// TIA Portal V20 export
FUNCTION "Level_Sim" : Void   // FC1, FBD
{ S7_Optimized_Access := 'TRUE' }
// stored: SetENOAutomatically false
BEGIN

REGION Network 1: LevelSimulation
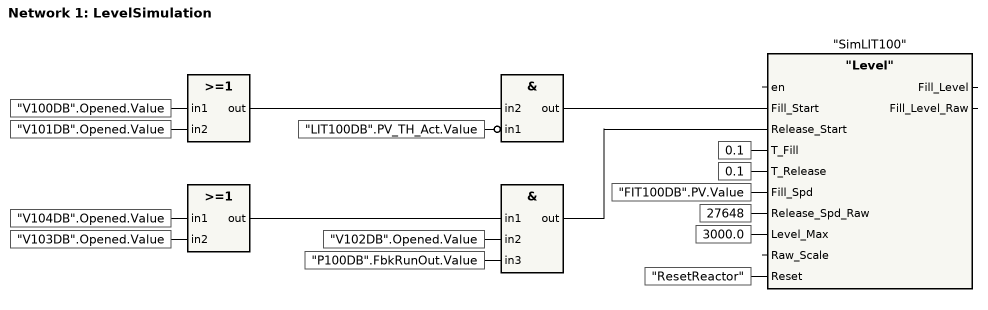
   "SimLIT100"(Fill_Start := ("V100DB".Opened.Value OR "V101DB".Opened.Value) AND NOT "LIT100DB".PV_TH_Act.Value,   // "Level"
               Release_Start := ("V104DB".Opened.Value OR "V103DB".Opened.Value) AND "V102DB".Opened.Value AND "P100DB".FbkRunOut.Value,
               T_Fill := 0.1,
               T_Release := 0.1,
               Fill_Spd := "FIT100DB".PV.Value,
               Release_Spd_Raw := 27648,
               Level_Max := 3000.0,
               Reset := "ResetReactor");
END_REGION
END_FUNCTION
